{attribute 'linkalways'} 
{attribute 'no_explicit_call' := 'This FB is a CLASS and must be accessed using methods or properties'}
{attribute 'enable_dynamic_creation'}
FUNCTION_BLOCK FINAL DigitalInputNode EXTENDS Node
VAR
	input AT %I* : BOOL;
	out : _BOOL(FALSE);
END_VAR

METHOD PUBLIC Clone : I_Node
VAR
END_VAR
Clone := this^;
END_METHOD

METHOD Dispose
VAR_INPUT
END_VAR
END_METHOD

METHOD FB_init : BOOL
VAR_INPUT
	bInitRetains : BOOL; // if TRUE, the retain variables are initialized (warm start / cold start)
	bInCopyCode : BOOL;  // if TRUE, the instance afterwards gets moved into the copy code (online change)
END_VAR
AddOutput('out', out);
END_METHOD

METHOD PROTECTED OnExecute : HRESULT
VAR
END_VAR
out.value := input;
END_METHOD

END_FUNCTION_BLOCK

(* stored: Version 1.1.0.1, ProductVersion 3.1.4024.12
   POU DigitalInputNode: Id {0dd4bd2b-0bb5-4458-a128-d5a89ab0178d}, SpecialFunc None
   Folder Constructor: Id {05b25e99-5c4d-4f85-b600-38bc711952f5}
   Method Clone: Id {1c79340a-7049-46d3-82de-091d1fd1a902}
   Method Dispose: Id {a14daa47-c044-4244-9f75-072ac12a55d0}
   Method FB_init: Id {d97e36ef-3322-46e9-b125-9ee1f29d291c}
   Method OnExecute: Id {c212795b-274d-4520-8ab4-0c7f2f195a63} *)
